FUNCTION_BLOCK Account

VAR
        PRIVATE 
             lrBalance : LREAL := 0.0; 
		END_VAR
END_VAR

METHOD PUBLIC Deposit : BOOL
VAR_INPUT
    lrAmount : LREAL;
END_VAR
IF lrAmount > 0 THEN
    lrBalance := lrBalance + lrAmount;
    Deposit := TRUE;
ELSE
    Deposit := FALSE;
END_IF
END_METHOD

END_FUNCTION_BLOCK

(* stored: Version 1.1.0.1, ProductVersion 3.1.4024.16
   POU Account: Id {ec5a15dd-b1f1-40e0-b446-f833c3745b63}, SpecialFunc None
   Method Deposit: Id {f530cf4a-1f11-41cf-8f3d-3f217829e74f} *)
